% RSLogix 500 project P8_KOBIERSKI_M.RSS, saved by version 8.30.00.16 %
PROJECT "UNTITLED"    % processor: Bul.1763 MicroLogix 1100 Series B %

PROGRAM FILES
  LAD 2 "MAIN"  3 rungs
  LAD 3 "IO"  3 rungs
  LAD 4 "CTRL"  12 rungs

DATA FILES
  O0 OUTPUT  4 elements
  I1 INPUT  6 elements
  S2 STATUS  66 elements
  B3 BINARY  1 elements
  T4 TIMER  1 elements
  C5 COUNTER  1 elements
  R6 CONTROL  1 elements
  N7 INTEGER  8 elements
  F8 FLOAT  2 elements

LADDER 2 "MAIN"
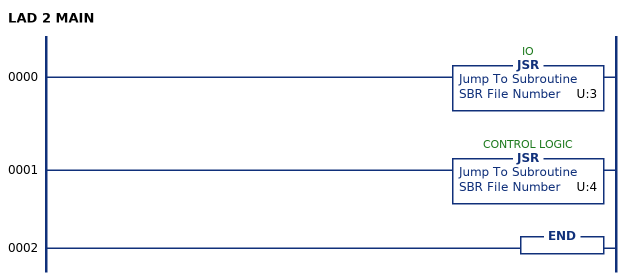
% Rung: 0 %
SOR JSR U:3 EOR
%   U:3  "IO" %
% Rung: 1 %
SOR JSR U:4 EOR
%   U:4  "CONTROL LOGIC" %
% Rung: 2 %
SOR END EOR

LADDER 3 "IO"
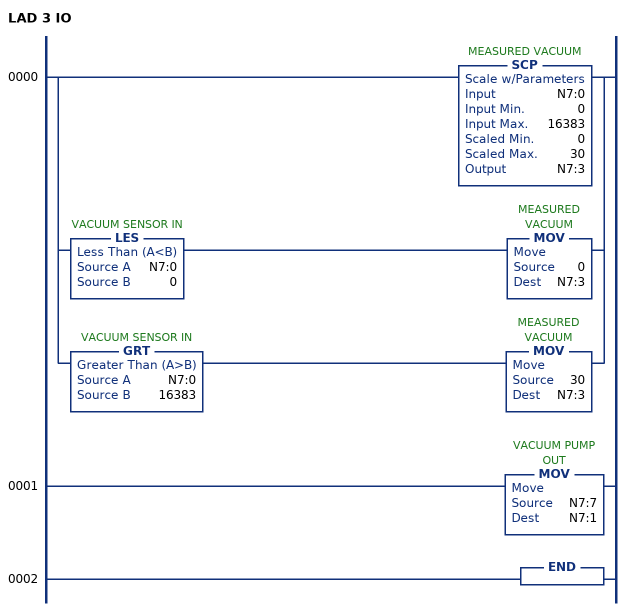
% Rung: 0 %
SOR BST SCP N7:0 0 16383 0 30 N7:3 NXB LES N7:0 0 MOV 0 N7:3 NXB GRT N7:0 16383 MOV 30 N7:3 BND EOR
%   N7:0  "VACUUM SENSOR IN" %
%   N7:3  "MEASURED VACUUM" %
% Rung: 1 %
SOR MOV N7:7 N7:1 EOR
%   N7:7  "NEW VACUUM PUMP SETPOINT" %
%   N7:1  "VACUUM PUMP OUT" %
% Rung: 2 %
SOR END EOR

LADDER 4 "CTRL"
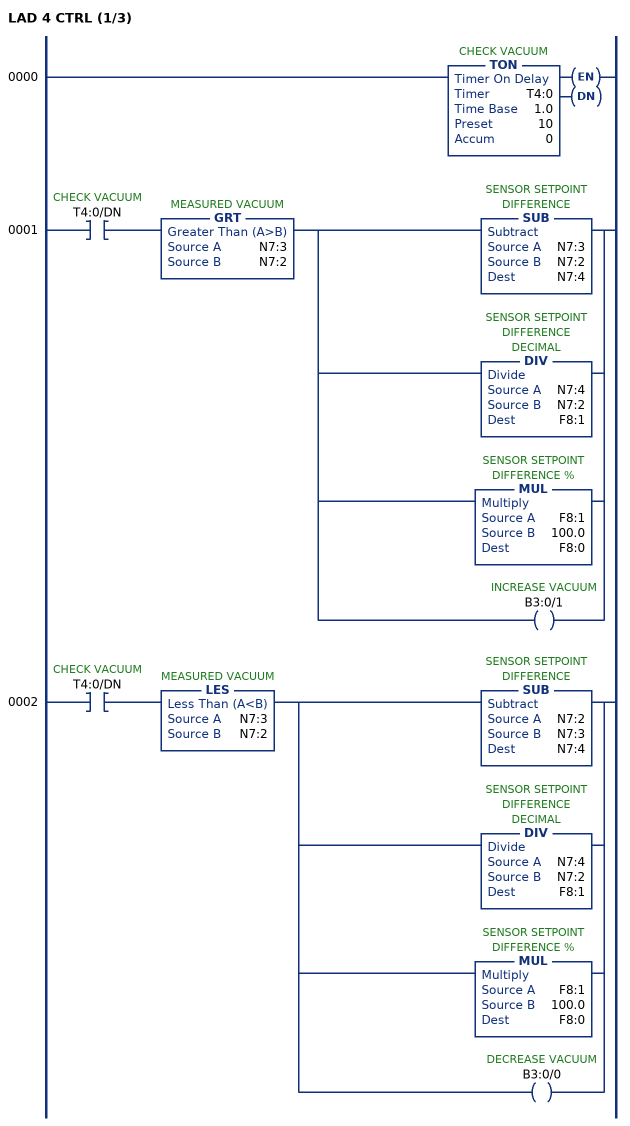
% Rung: 0 %
SOR TON T4:0 1.0 10 0 EOR
%   T4:0  "CHECK VACUUM" %
% Rung: 1 %
SOR XIC T4:0/DN GRT N7:3 N7:2 BST SUB N7:3 N7:2 N7:4 NXB DIV N7:4 N7:2 F8:1 NXB MUL F8:1 100.0 F8:0 NXB OTE B3:0/1 BND EOR
%   T4:0  "CHECK VACUUM" %
%   N7:3  "MEASURED VACUUM" %
%   N7:2  "VACUUM SETPOINT" %
%   N7:4  "SENSOR SETPOINT DIFFERENCE" %
%   F8:1  "SENSOR SETPOINT DIFFERENCE DECIMAL" %
%   F8:0  "SENSOR SETPOINT DIFFERENCE %" %
%   B3:0/1  "INCREASE VACUUM" %
% Rung: 2 %
SOR XIC T4:0/DN LES N7:3 N7:2 BST SUB N7:2 N7:3 N7:4 NXB DIV N7:4 N7:2 F8:1 NXB MUL F8:1 100.0 F8:0 NXB OTE B3:0/0 BND EOR
%   T4:0  "CHECK VACUUM" %
%   N7:3  "MEASURED VACUUM" %
%   N7:2  "VACUUM SETPOINT" %
%   N7:4  "SENSOR SETPOINT DIFFERENCE" %
%   F8:1  "SENSOR SETPOINT DIFFERENCE DECIMAL" %
%   F8:0  "SENSOR SETPOINT DIFFERENCE %" %
%   B3:0/0  "DECREASE VACUUM" %

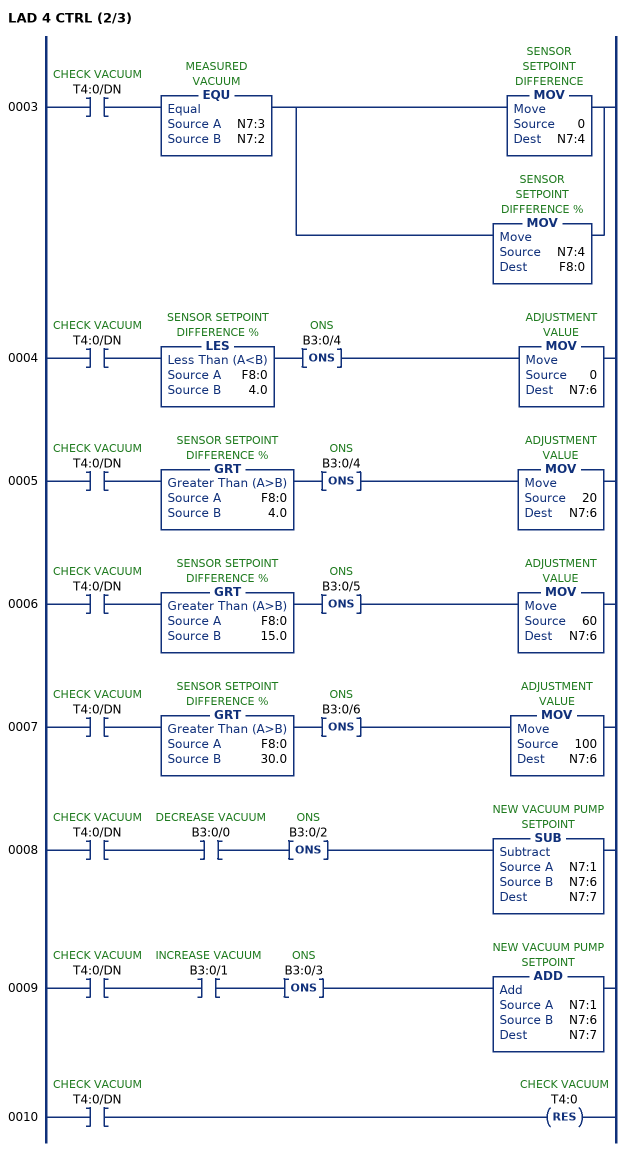
% Rung: 3 %
SOR XIC T4:0/DN EQU N7:3 N7:2 BST MOV 0 N7:4 NXB MOV N7:4 F8:0 BND EOR
%   T4:0  "CHECK VACUUM" %
%   N7:3  "MEASURED VACUUM" %
%   N7:2  "VACUUM SETPOINT" %
%   N7:4  "SENSOR SETPOINT DIFFERENCE" %
%   F8:0  "SENSOR SETPOINT DIFFERENCE %" %
% Rung: 4 %
SOR XIC T4:0/DN LES F8:0 4.0 ONS B3:0/4 MOV 0 N7:6 EOR
%   T4:0  "CHECK VACUUM" %
%   F8:0  "SENSOR SETPOINT DIFFERENCE %" %
%   B3:0/4  "ONS" %
%   N7:6  "ADJUSTMENT VALUE" %
% Rung: 5 %
SOR XIC T4:0/DN GRT F8:0 4.0 ONS B3:0/4 MOV 20 N7:6 EOR
%   T4:0  "CHECK VACUUM" %
%   F8:0  "SENSOR SETPOINT DIFFERENCE %" %
%   B3:0/4  "ONS" %
%   N7:6  "ADJUSTMENT VALUE" %
% Rung: 6 %
SOR XIC T4:0/DN GRT F8:0 15.0 ONS B3:0/5 MOV 60 N7:6 EOR
%   T4:0  "CHECK VACUUM" %
%   F8:0  "SENSOR SETPOINT DIFFERENCE %" %
%   B3:0/5  "ONS" %
%   N7:6  "ADJUSTMENT VALUE" %
% Rung: 7 %
SOR XIC T4:0/DN GRT F8:0 30.0 ONS B3:0/6 MOV 100 N7:6 EOR
%   T4:0  "CHECK VACUUM" %
%   F8:0  "SENSOR SETPOINT DIFFERENCE %" %
%   B3:0/6  "ONS" %
%   N7:6  "ADJUSTMENT VALUE" %
% Rung: 8 %
SOR XIC T4:0/DN XIC B3:0/0 ONS B3:0/2 SUB N7:1 N7:6 N7:7 EOR
%   T4:0  "CHECK VACUUM" %
%   B3:0/0  "DECREASE VACUUM" %
%   B3:0/2  "ONS" %
%   N7:1  "VACUUM PUMP OUT" %
%   N7:6  "ADJUSTMENT VALUE" %
%   N7:7  "NEW VACUUM PUMP SETPOINT" %
% Rung: 9 %
SOR XIC T4:0/DN XIC B3:0/1 ONS B3:0/3 ADD N7:1 N7:6 N7:7 EOR
%   T4:0  "CHECK VACUUM" %
%   B3:0/1  "INCREASE VACUUM" %
%   B3:0/3  "ONS" %
%   N7:1  "VACUUM PUMP OUT" %
%   N7:6  "ADJUSTMENT VALUE" %
%   N7:7  "NEW VACUUM PUMP SETPOINT" %
% Rung: 10 %
SOR XIC T4:0/DN RES T4:0 EOR
%   T4:0  "CHECK VACUUM" %

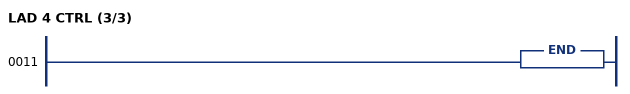
% Rung: 11 %
SOR END EOR

DATA TABLE (non-zero values as saved)
DATA T4
% .PRE .ACC %
% T4:0 % 10 0
DATA N7
% N7:0 % 0 0 15 0 0 0 0 0
